// TIA Portal V20 export
DATA_BLOCK "SimpleEnc_DB"   // DB39
// stored: InstanceOfName SimpleEnc, InstanceOfType FB
"SimpleEnc"
   // VAR_INPUT
   //    position : DInt;
   //    init : Bool;
   // END_VAR
   // VAR_IN_OUT
   //    tel81 : PD_TEL81;
   // END_VAR
   // VAR
   //    statError : Bool;
   //    statOldPos : DInt;
   // END_VAR
BEGIN
END_DATA_BLOCK
